// TIA Portal V20 export
TYPE "LBP_typeInternal3"
TITLE = Internal data type for basic program / Type de données interne pour programme de base
// Data type only for internal use in the basic program / Type de données réservé à l'utilisation interne dans le programme de base
   STRUCT
      "Version" { ExternalAccessible := 'False'; ExternalVisible := 'False'; ExternalWritable := 'False'} : UDInt;
      BlockReturnValue { ExternalAccessible := 'False'; ExternalVisible := 'False'; ExternalWritable := 'False'} : UDInt;
      AlarmList { ExternalAccessible := 'False'; ExternalVisible := 'False'; ExternalWritable := 'False'} : Array[1..6] of Struct
         ARID : UInt;
         AlarmMessage : Bool;
         OperationMessage : Bool;
         AlarmIsComing : Bool;
         StopPlc : Bool;
         NumberOfExtendedValues : USInt;
         AlarmNumber : UDInt;
         ExtendedValueList : Array[1..9] of UDInt;
      END_STRUCT;
   END_STRUCT;
END_TYPE
